FUNCTION_BLOCK TestPostLogChain
VAR_IN_OUT
	logBuffer : LogBuffer;
END_VAR
VAR_OUTPUT
END_VAR
VAR
	await: Await;
	step: UDINT; 
	
	client: FB_IotHttpClient := (
		sHostName:='localhost',
		bKeepAlive:=TRUE,
		tConnectionTimeout:=T#10S,
		nHostPort:=8000
	);
	
	request: FB_IotHttpRequest;
	endpoint: STRING := '/log';
	
	fbJson: FB_JsonDomParser;
	jsonDoc: SJsonValue;
	
	json: Json;
	risingEdge: R_TRIG;
	send: BOOL;
	requestOperation: BOOL;
	
	logMessage : STRING(255);

	// Callbacks
	onRequestError : OnRequestError:= (errorName:='TestPostLogChain.OnRequestError', onErrorStep:=500);
	resetStepOnSuccess: StepChainResetter := (stepReference:=step);  
END_VAR
VAR CONSTANT
	cMax : INT := 100;
END_VAR

risingEdge(CLK:=send );
client.Execute();

CASE step OF 
	
	000: // Basic init step
	
		await.continueIf(client.bConfigured AND logBuffer.pop(logMessage));
		
	010:
		
		json.create(logMessage);
		requestOperation := request.SendRequest(
			sUri:= '/log', 
			fbClient:= client, 
			eRequestType:= ETcIotHttpRequestType.HTTP_POST, 
			pContent:= ADR(json.payload), 			
			nContentSize:= len2(ADR(json.payload)), 
			0
		);
		
		await.evalue(requestOperation, resetStepOnSuccess, onRequestError, 'Error during request');

		
END_CASE

METHOD FB_init : BOOL
VAR_INPUT
	bInitRetains : BOOL; // if TRUE, the retain variables are initialized (warm start / cold start)
	bInCopyCode : BOOL;  // if TRUE, the instance afterwards gets moved into the copy code (online change)
END_VAR
await.setStepPointer := ADR(step);
await.setIncreaseValue := 10;
END_METHOD

END_FUNCTION_BLOCK

(* stored: Version 1.1.0.1, ProductVersion 3.1.4024.12
   POU TestPostLogChain: Id {157a5f80-8dfd-4678-859e-1462e0d7b71a}, SpecialFunc None
   Method FB_init: Id {de411cd0-4760-4b28-a254-913b98e98a42} *)
